Omron CX-Programmer project NewProject (CX-Programmer 9.75)

# PLC NewPLC1: CP1L M

## Global symbols (name address type ; comment)
0.00 BOOL  ; START
0.01 BOOL  ; STOP
A354 CHANNEL  ; HARI KE -
D0 CHANNEL  ; DETIK
D1 CHANNEL  ; MENIT
D2 CHANNEL  ; JAM
D3 CHANNEL  ; TANGGAL
D4 CHANNEL  ; BULAN
D5 CHANNEL  ; TAHUN
W0.01 BOOL  ; SENIN - JUM'AT
W0.02 BOOL  ; 08:00 - 17:00
W0.03 BOOL  ; OFF
test _INV201_ReadParameter

## Program NewProgram1 (cyclic task 0)

### Section Section1

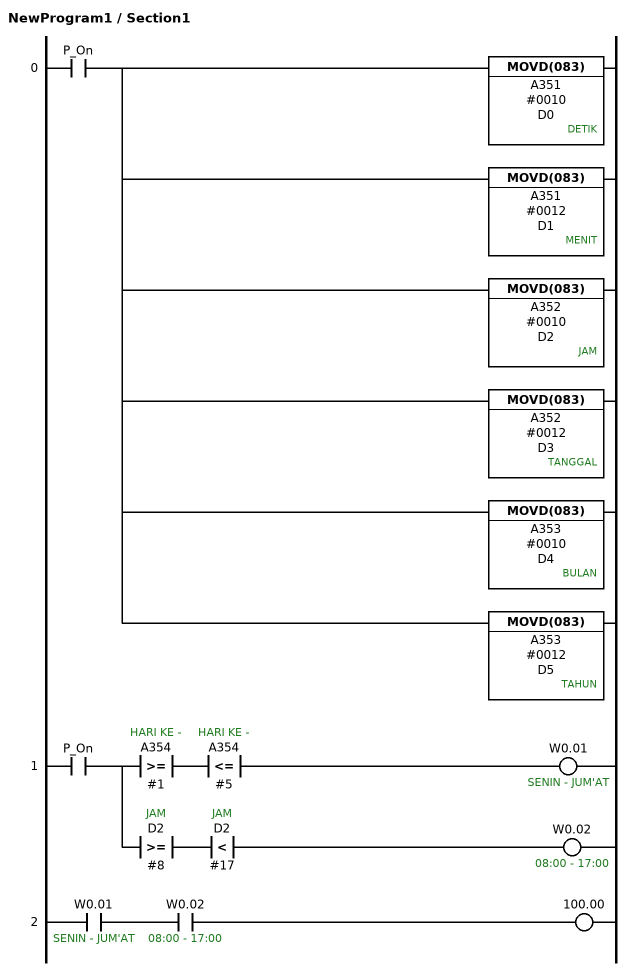
; rung 0
LD P_On
MOVD(083) A351 #0010 D0  ; DETIK
MOVD(083) A351 #0012 D1  ; MENIT
MOVD(083) A352 #0010 D2  ; JAM
MOVD(083) A352 #0012 D3  ; TANGGAL
MOVD(083) A353 #0010 D4  ; BULAN
MOVD(083) A353 #0012 D5  ; TAHUN
; rung 1
LD P_On
OUT TR0
AND>=(325) A354 #1  ; HARI KE -
AND<=(315) A354 #5  ; HARI KE -
OUT W0.01  ; SENIN - JUM'AT
LD TR0
AND>=(325) D2 #8  ; JAM
AND<(310) D2 #17  ; JAM
OUT W0.02  ; 08:00 - 17:00
; rung 2
LD W0.01  ; SENIN - JUM'AT
AND W0.02  ; 08:00 - 17:00
OUT 100.00

### Section END
; rung 0
END(001)

## Function block _INV201_ReadParameter (Omron library block, body left out)